{attribute addProperty BoxType "KL2819"}
{attribute addProperty Id "StatusAT %I*USINT000DiagAT %I*WORD000CtrlAT %Q*USINT000OutputAT %Q*WORD000"}
{attribute addProperty CRC "2037047455"}
{attribute addProperty SizeInBites "0"}
{attribute addProperty SizeInBytes "0"}
TYPE Channel_796AE09F :
STRUCT
	{attribute addProperty Name "Status"}
	Status AT %I* : USINT;
	{attribute addProperty Name "Diag"}
	Diag AT %I* : WORD;
	{attribute addProperty Name "Ctrl"}
	Ctrl AT %Q* : USINT;
	{attribute addProperty Name "Output"}
	Output AT %Q* : WORD;
END_STRUCT
END_TYPE

(* stored: Version 1.2.0.0, ProductVersion 3.1.4024.9
   DUT Channel_796AE09F: Id {cb647f17-4bdb-4872-9315-1d01ba410e0c} *)
